FUNCTION_BLOCK FB_Observer_BYTE EXTENDS FB_AbstractObserver
VAR
    _nVal:              BYTE;
END_VAR

METHOD FB_init : BOOL
VAR_INPUT
	bInitRetains : BOOL; // if TRUE, the retain variables are initialized (warm start / cold start)
	bInCopyCode : BOOL;  // if TRUE, the instance afterwards gets moved into the copy code (online change)
END_VAR
THIS^._nTypeClass := __SYSTEM.TYPE_CLASS.TYPE_BYTE;
THIS^._pVal := ADR(THIS^._nVal);
THIS^._nSize := SIZEOF(THIS^._nVal);
END_METHOD

PROPERTY nValue8 : BYTE
GET
nValue8 := THIS^._nVal;
END_GET
END_PROPERTY

END_FUNCTION_BLOCK

(* stored: Version 1.1.0.1, ProductVersion 3.1.4024.12
   POU FB_Observer_BYTE: Id {181a47c5-b9d3-0b6c-3efd-0fee4a8fc405}, SpecialFunc None
   Method FB_init: Id {264c6655-43ce-0f7b-1f63-bd94a34cf0ad}
   Property nValue8: Id {84bcd076-87eb-0ad7-1361-db806e34c38e}
   Get Get: Id {3413ef97-cf5f-0f27-02c7-f1179c5ca886} *)
